// TIA Portal V16 export
// export: Created 2023-08-28T09:37:42.2517903Z, ExportSetting WithDefaults, DisplayName Totally Integrated Automation Portal, DisplayVersion V16 Update 6, DisplayName TIA Portal Version Control Interface, DisplayVersion V16 Update 2, DisplayName TIA Portal Openness, DisplayVersion V16 Update 6, DisplayName STEP 7 Professional, DisplayVersion V16 Update 6, DisplayName STEP 7 Safety, DisplayVersion V16, DisplayName WinCC Advanced, DisplayVersion V16 Update 6
FUNCTION_BLOCK "06_M_Main and auxiliary pump"   // FB9, LAD
TITLE = Funkcja ustalająca napęd wiodący i dodatkowe
{ S7_Optimized_Access := 'TRUE' }
AUTHOR : rtecmer
VERSION : 0.1
// Ustalanie silnika wiodącego i dodatkowego następuje po sprawdzeniu czy dany napęd załączony jes na falownik czy na sieć. Procedura rozpoczyna się od ustalenia napędu wiodącego.
// stored: AutoNumber true, IsIECCheckEnabled false, IsRetainMemResEnabled false, MemoryReserve 500, SetENOAutomatically false, UDAEnableTagReadback false
   VAR_IN_OUT
      set_Motor2 : Bool;   // pomocniczy bit ustawiania pompę dodatkową nr1
      set_Motor3 : Bool;   // pomocniczy bit ustawiania pompę dodatkową nr2
      set_Motor4 : Bool;   // pomocniczy bit ustawiania pompę dodatkową nr3
   END_VAR
   VAR_TEMP
      tmp_Res_Motor2 : Bool;   // pomocniczy bit kasowania znacznika dodatkowej nr1
      tmp_Res_Motor3 : Bool;   // pomocniczy bit kasowania znacznika dodatkowej nr2
      tmp_Res_Motor4 : Bool;   // pomocniczy bit kasowania znacznika dodatkowej nr3
   END_VAR
   VAR_TEMP   // added for the SCL form of the ladder/FBD networks
      _w1 : Bool;
      _w2 : Bool;
      _w3 : Bool;
      _w4 : Bool;
      _w5 : Bool;
      _w6 : Bool;
   END_VAR
BEGIN

REGION Network 1: Znacznik pompy wiodącej
   // M218.0 - bit ustalający pompy wiodącą . Przekazywany do zmiennych "IN" funkcji  "Control of   Inverters"
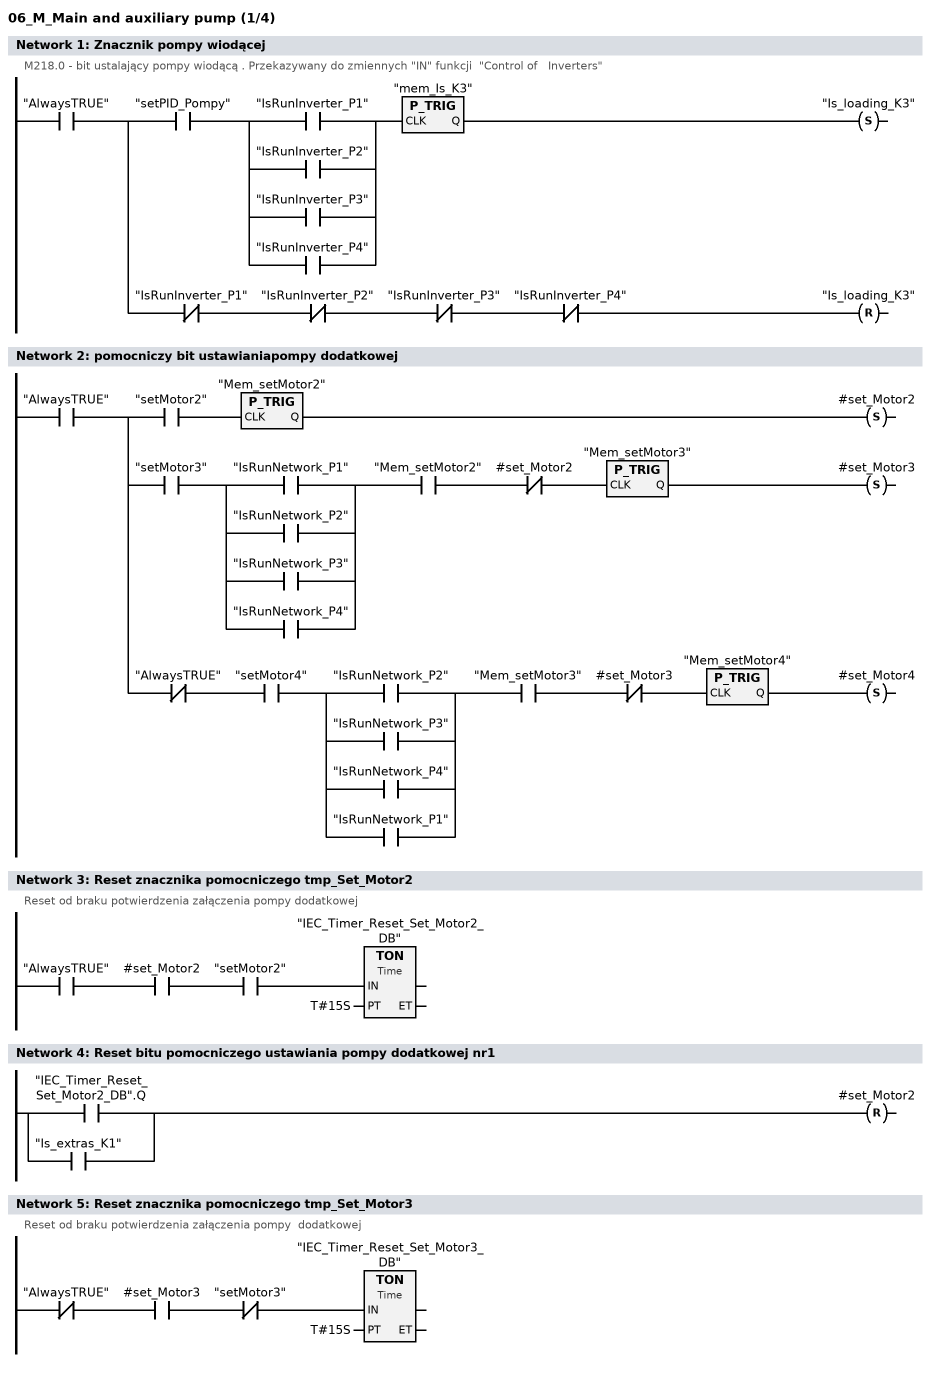
   RUNG wire#powerrail
      Contact( "AlwaysTRUE" )
      wire#w1
      Contact( "setPID_Pompy" )
      wire#w2
      Contact( "IsRunInverter_P1" )
      wire#w3
      P_Trig( "mem_Is_K3" )
      S_Coil( "Is_loading_K3" )
   END_RUNG
   RUNG wire#w2
      Contact( "IsRunInverter_P2" )
   END_RUNG wire#w3
   RUNG wire#w2
      Contact( "IsRunInverter_P3" )
   END_RUNG wire#w3
   RUNG wire#w2
      Contact( "IsRunInverter_P4" )
   END_RUNG wire#w3
   RUNG wire#w1
      I_Contact( "IsRunInverter_P1" )
      I_Contact( "IsRunInverter_P2" )
      I_Contact( "IsRunInverter_P3" )
      I_Contact( "IsRunInverter_P4" )
      R_Coil( "Is_loading_K3" )
   END_RUNG
   // the same network as SCL:
   #_w1 := "AlwaysTRUE" AND "setPID_Pompy" AND ("IsRunInverter_P1" OR "IsRunInverter_P2" OR "IsRunInverter_P3" OR "IsRunInverter_P4");
   #_w2 := #_w1 AND NOT "mem_Is_K3";   // rising edge
   "mem_Is_K3" := #_w1;
   IF #_w2 THEN "Is_loading_K3" := TRUE; END_IF;
   IF "AlwaysTRUE" AND NOT "IsRunInverter_P1" AND NOT "IsRunInverter_P2" AND NOT "IsRunInverter_P3" AND NOT "IsRunInverter_P4" THEN
       "Is_loading_K3" := FALSE;
   END_IF;
END_REGION

REGION Network 2: pomocniczy bit ustawianiapompy dodatkowej
   RUNG wire#powerrail
      Contact( "AlwaysTRUE" )
      wire#w1
      Contact( "setMotor2" )
      P_Trig( "Mem_setMotor2" )
      S_Coil( #set_Motor2 )
   END_RUNG
   RUNG wire#w1
      Contact( "setMotor3" )
      wire#w2
      Contact( "IsRunNetwork_P1" )
      wire#w3
      Contact( "Mem_setMotor2" )
      I_Contact( #set_Motor2 )
      P_Trig( "Mem_setMotor3" )
      S_Coil( #set_Motor3 )
   END_RUNG
   RUNG wire#w2
      Contact( "IsRunNetwork_P2" )
   END_RUNG wire#w3
   RUNG wire#w2
      Contact( "IsRunNetwork_P3" )
   END_RUNG wire#w3
   RUNG wire#w2
      Contact( "IsRunNetwork_P4" )
   END_RUNG wire#w3
   RUNG wire#w1
      I_Contact( "AlwaysTRUE" )
      Contact( "setMotor4" )
      wire#w4
      Contact( "IsRunNetwork_P2" )
      wire#w5
      Contact( "Mem_setMotor3" )
      I_Contact( #set_Motor3 )
      P_Trig( "Mem_setMotor4" )
      S_Coil( #set_Motor4 )
   END_RUNG
   RUNG wire#w4
      Contact( "IsRunNetwork_P3" )
   END_RUNG wire#w5
   RUNG wire#w4
      Contact( "IsRunNetwork_P4" )
   END_RUNG wire#w5
   RUNG wire#w4
      Contact( "IsRunNetwork_P1" )
   END_RUNG wire#w5
   // the same network as SCL:
   #_w1 := "AlwaysTRUE" AND "setMotor2";
   #_w2 := #_w1 AND NOT "Mem_setMotor2";   // rising edge
   "Mem_setMotor2" := #_w1;
   IF #_w2 THEN #set_Motor2 := TRUE; END_IF;
   #_w3 := "AlwaysTRUE" AND "setMotor3" AND ("IsRunNetwork_P1" OR "IsRunNetwork_P2" OR "IsRunNetwork_P3" OR "IsRunNetwork_P4") AND "Mem_setMotor2" AND NOT #set_Motor2;
   #_w4 := #_w3 AND NOT "Mem_setMotor3";   // rising edge
   "Mem_setMotor3" := #_w3;
   IF #_w4 THEN #set_Motor3 := TRUE; END_IF;
   #_w5 := "AlwaysTRUE" AND NOT "AlwaysTRUE" AND "setMotor4" AND ("IsRunNetwork_P2" OR "IsRunNetwork_P3" OR "IsRunNetwork_P4" OR "IsRunNetwork_P1") AND "Mem_setMotor3" AND NOT #set_Motor3;
   #_w6 := #_w5 AND NOT "Mem_setMotor4";   // rising edge
   "Mem_setMotor4" := #_w5;
   IF #_w6 THEN #set_Motor4 := TRUE; END_IF;
END_REGION

REGION Network 3: Reset znacznika pomocniczego tmp_Set_Motor2
   // Reset od braku potwierdzenia załączenia pompy dodatkowej
   RUNG wire#powerrail
      Contact( "AlwaysTRUE" )
      Contact( #set_Motor2 )
      Contact( "setMotor2" )
      { S7_Templates := "time_type := Time" } "IEC_Timer_Reset_Set_Motor2_DB".TON(pt := T#15S, et =>)
   END_RUNG
   // the same network as SCL:
   "IEC_Timer_Reset_Set_Motor2_DB".TON(IN := "AlwaysTRUE" AND #set_Motor2 AND "setMotor2", PT := T#15S);
END_REGION

REGION Network 4: Reset bitu pomocniczego ustawiania pompy dodatkowej nr1
   RUNG wire#powerrail
      Contact( "IEC_Timer_Reset_Set_Motor2_DB".Q )
      wire#w1
      R_Coil( #set_Motor2 )
   END_RUNG
   RUNG wire#powerrail
      Contact( "Is_extras_K1" )
   END_RUNG wire#w1
   // the same network as SCL:
   IF "IEC_Timer_Reset_Set_Motor2_DB".Q OR "Is_extras_K1" THEN #set_Motor2 := FALSE; END_IF;
END_REGION

REGION Network 5: Reset znacznika pomocniczego tmp_Set_Motor3
   // Reset od braku potwierdzenia załączenia pompy  dodatkowej
   RUNG wire#powerrail
      I_Contact( "AlwaysTRUE" )
      Contact( #set_Motor3 )
      I_Contact( "setMotor3" )
      { S7_Templates := "time_type := Time" } "IEC_Timer_Reset_Set_Motor3_DB".TON(pt := T#15S, et =>)
   END_RUNG
   // the same network as SCL:
   "IEC_Timer_Reset_Set_Motor3_DB".TON(IN := NOT "AlwaysTRUE" AND #set_Motor3 AND NOT "setMotor3", PT := T#15S);
END_REGION

REGION Network 6: Reset pomocniczego bit ustawianiapompy dodatkowej nr2
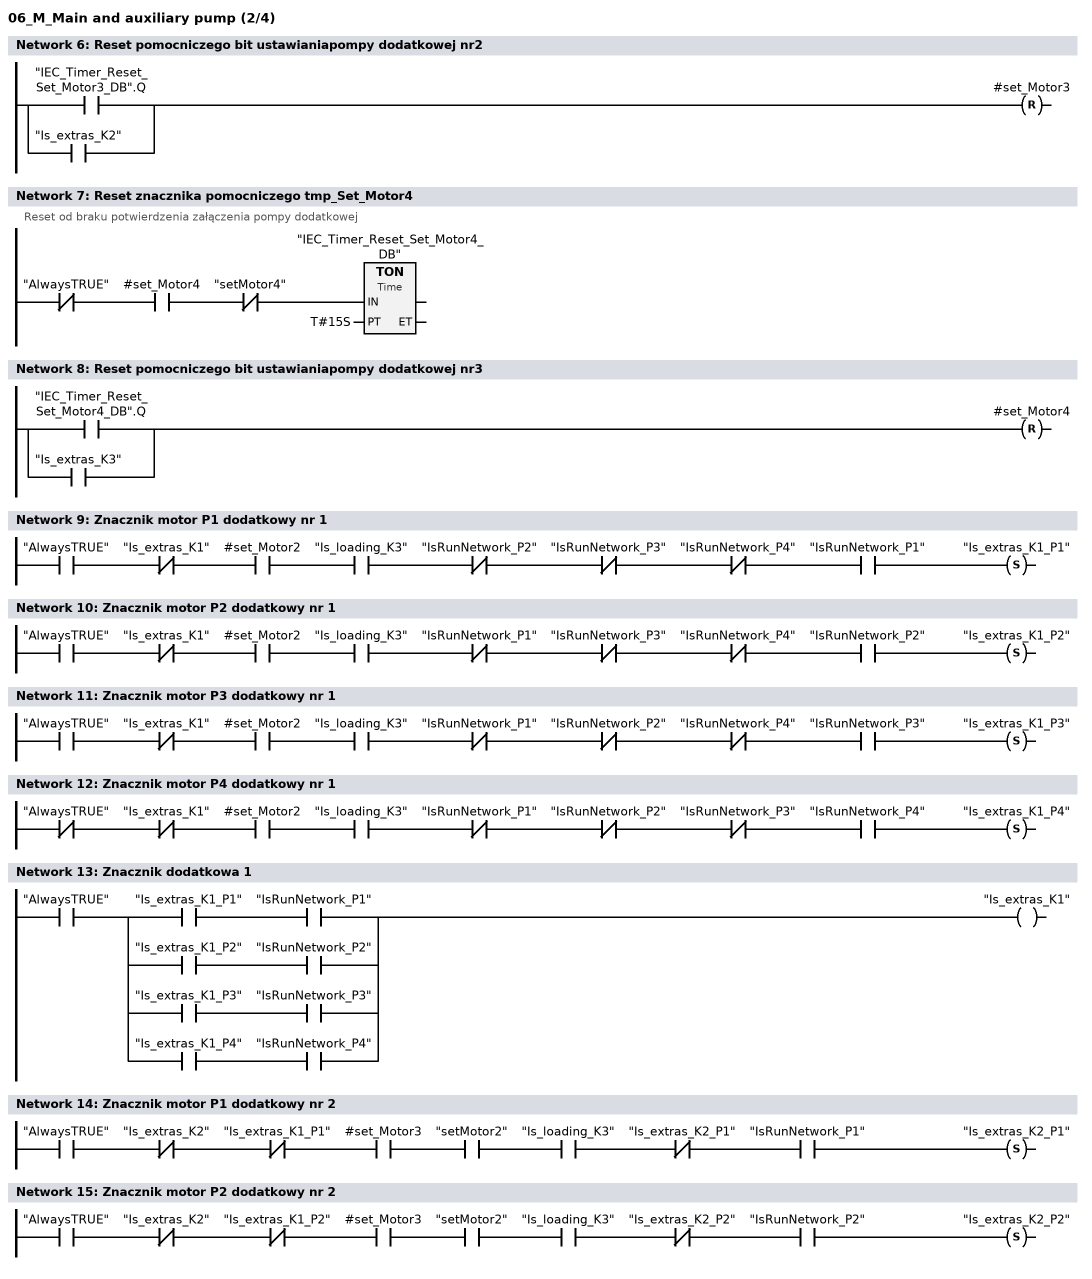
   RUNG wire#powerrail
      Contact( "IEC_Timer_Reset_Set_Motor3_DB".Q )
      wire#w1
      R_Coil( #set_Motor3 )
   END_RUNG
   RUNG wire#powerrail
      Contact( "Is_extras_K2" )
   END_RUNG wire#w1
   // the same network as SCL:
   IF "IEC_Timer_Reset_Set_Motor3_DB".Q OR "Is_extras_K2" THEN #set_Motor3 := FALSE; END_IF;
END_REGION

REGION Network 7: Reset znacznika pomocniczego tmp_Set_Motor4
   // Reset od braku potwierdzenia załączenia pompy dodatkowej
   RUNG wire#powerrail
      I_Contact( "AlwaysTRUE" )
      Contact( #set_Motor4 )
      I_Contact( "setMotor4" )
      { S7_Templates := "time_type := Time" } "IEC_Timer_Reset_Set_Motor4_DB".TON(pt := T#15S, et =>)
   END_RUNG
   // the same network as SCL:
   "IEC_Timer_Reset_Set_Motor4_DB".TON(IN := NOT "AlwaysTRUE" AND #set_Motor4 AND NOT "setMotor4", PT := T#15S);
END_REGION

REGION Network 8: Reset pomocniczego bit ustawianiapompy dodatkowej nr3
   RUNG wire#powerrail
      Contact( "IEC_Timer_Reset_Set_Motor4_DB".Q )
      wire#w1
      R_Coil( #set_Motor4 )
   END_RUNG
   RUNG wire#powerrail
      Contact( "Is_extras_K3" )
   END_RUNG wire#w1
   // the same network as SCL:
   IF "IEC_Timer_Reset_Set_Motor4_DB".Q OR "Is_extras_K3" THEN #set_Motor4 := FALSE; END_IF;
END_REGION

REGION Network 9: Znacznik motor P1 dodatkowy nr 1
   RUNG wire#powerrail
      Contact( "AlwaysTRUE" )
      I_Contact( "Is_extras_K1" )
      Contact( #set_Motor2 )
      Contact( "Is_loading_K3" )
      I_Contact( "IsRunNetwork_P2" )
      I_Contact( "IsRunNetwork_P3" )
      I_Contact( "IsRunNetwork_P4" )
      Contact( "IsRunNetwork_P1" )
      S_Coil( "Is_extras_K1_P1" )
   END_RUNG
   // the same network as SCL:
   IF "AlwaysTRUE" AND NOT "Is_extras_K1" AND #set_Motor2 AND "Is_loading_K3" AND NOT "IsRunNetwork_P2" AND NOT "IsRunNetwork_P3" AND NOT "IsRunNetwork_P4" AND "IsRunNetwork_P1" THEN
       "Is_extras_K1_P1" := TRUE;
   END_IF;
END_REGION

REGION Network 10: Znacznik motor P2 dodatkowy nr 1
   RUNG wire#powerrail
      Contact( "AlwaysTRUE" )
      I_Contact( "Is_extras_K1" )
      Contact( #set_Motor2 )
      Contact( "Is_loading_K3" )
      I_Contact( "IsRunNetwork_P1" )
      I_Contact( "IsRunNetwork_P3" )
      I_Contact( "IsRunNetwork_P4" )
      Contact( "IsRunNetwork_P2" )
      S_Coil( "Is_extras_K1_P2" )
   END_RUNG
   // the same network as SCL:
   IF "AlwaysTRUE" AND NOT "Is_extras_K1" AND #set_Motor2 AND "Is_loading_K3" AND NOT "IsRunNetwork_P1" AND NOT "IsRunNetwork_P3" AND NOT "IsRunNetwork_P4" AND "IsRunNetwork_P2" THEN
       "Is_extras_K1_P2" := TRUE;
   END_IF;
END_REGION

REGION Network 11: Znacznik motor P3 dodatkowy nr 1
   RUNG wire#powerrail
      Contact( "AlwaysTRUE" )
      I_Contact( "Is_extras_K1" )
      Contact( #set_Motor2 )
      Contact( "Is_loading_K3" )
      I_Contact( "IsRunNetwork_P1" )
      I_Contact( "IsRunNetwork_P2" )
      I_Contact( "IsRunNetwork_P4" )
      Contact( "IsRunNetwork_P3" )
      S_Coil( "Is_extras_K1_P3" )
   END_RUNG
   // the same network as SCL:
   IF "AlwaysTRUE" AND NOT "Is_extras_K1" AND #set_Motor2 AND "Is_loading_K3" AND NOT "IsRunNetwork_P1" AND NOT "IsRunNetwork_P2" AND NOT "IsRunNetwork_P4" AND "IsRunNetwork_P3" THEN
       "Is_extras_K1_P3" := TRUE;
   END_IF;
END_REGION

REGION Network 12: Znacznik motor P4 dodatkowy nr 1
   RUNG wire#powerrail
      I_Contact( "AlwaysTRUE" )
      I_Contact( "Is_extras_K1" )
      Contact( #set_Motor2 )
      Contact( "Is_loading_K3" )
      I_Contact( "IsRunNetwork_P1" )
      I_Contact( "IsRunNetwork_P2" )
      I_Contact( "IsRunNetwork_P3" )
      Contact( "IsRunNetwork_P4" )
      S_Coil( "Is_extras_K1_P4" )
   END_RUNG
   // the same network as SCL:
   IF NOT "AlwaysTRUE" AND NOT "Is_extras_K1" AND #set_Motor2 AND "Is_loading_K3" AND NOT "IsRunNetwork_P1" AND NOT "IsRunNetwork_P2" AND NOT "IsRunNetwork_P3" AND "IsRunNetwork_P4" THEN
       "Is_extras_K1_P4" := TRUE;
   END_IF;
END_REGION

REGION Network 13: Znacznik dodatkowa 1
   RUNG wire#powerrail
      Contact( "AlwaysTRUE" )
      wire#w1
      Contact( "Is_extras_K1_P1" )
      Contact( "IsRunNetwork_P1" )
      wire#w2
      Coil( "Is_extras_K1" )
   END_RUNG
   RUNG wire#w1
      Contact( "Is_extras_K1_P2" )
      Contact( "IsRunNetwork_P2" )
   END_RUNG wire#w2
   RUNG wire#w1
      Contact( "Is_extras_K1_P3" )
      Contact( "IsRunNetwork_P3" )
   END_RUNG wire#w2
   RUNG wire#w1
      Contact( "Is_extras_K1_P4" )
      Contact( "IsRunNetwork_P4" )
   END_RUNG wire#w2
   // the same network as SCL:
   "Is_extras_K1" := "AlwaysTRUE" AND (("Is_extras_K1_P1" AND "IsRunNetwork_P1") OR ("Is_extras_K1_P2" AND "IsRunNetwork_P2") OR ("Is_extras_K1_P3" AND "IsRunNetwork_P3") OR ("Is_extras_K1_P4" AND "IsRunNetwork_P4"));
END_REGION

REGION Network 14: Znacznik motor P1 dodatkowy nr 2
   RUNG wire#powerrail
      Contact( "AlwaysTRUE" )
      I_Contact( "Is_extras_K2" )
      I_Contact( "Is_extras_K1_P1" )
      Contact( #set_Motor3 )
      Contact( "setMotor2" )
      Contact( "Is_loading_K3" )
      I_Contact( "Is_extras_K2_P1" )
      Contact( "IsRunNetwork_P1" )
      S_Coil( "Is_extras_K2_P1" )
   END_RUNG
   // the same network as SCL:
   IF "AlwaysTRUE" AND NOT "Is_extras_K2" AND NOT "Is_extras_K1_P1" AND #set_Motor3 AND "setMotor2" AND "Is_loading_K3" AND NOT "Is_extras_K2_P1" AND "IsRunNetwork_P1" THEN
       "Is_extras_K2_P1" := TRUE;
   END_IF;
END_REGION

REGION Network 15: Znacznik motor P2 dodatkowy nr 2
   RUNG wire#powerrail
      Contact( "AlwaysTRUE" )
      I_Contact( "Is_extras_K2" )
      I_Contact( "Is_extras_K1_P2" )
      Contact( #set_Motor3 )
      Contact( "setMotor2" )
      Contact( "Is_loading_K3" )
      I_Contact( "Is_extras_K2_P2" )
      Contact( "IsRunNetwork_P2" )
      S_Coil( "Is_extras_K2_P2" )
   END_RUNG
   // the same network as SCL:
   IF "AlwaysTRUE" AND NOT "Is_extras_K2" AND NOT "Is_extras_K1_P2" AND #set_Motor3 AND "setMotor2" AND "Is_loading_K3" AND NOT "Is_extras_K2_P2" AND "IsRunNetwork_P2" THEN
       "Is_extras_K2_P2" := TRUE;
   END_IF;
END_REGION

REGION Network 16: Znacznik motor P3 dodatkowy nr 2
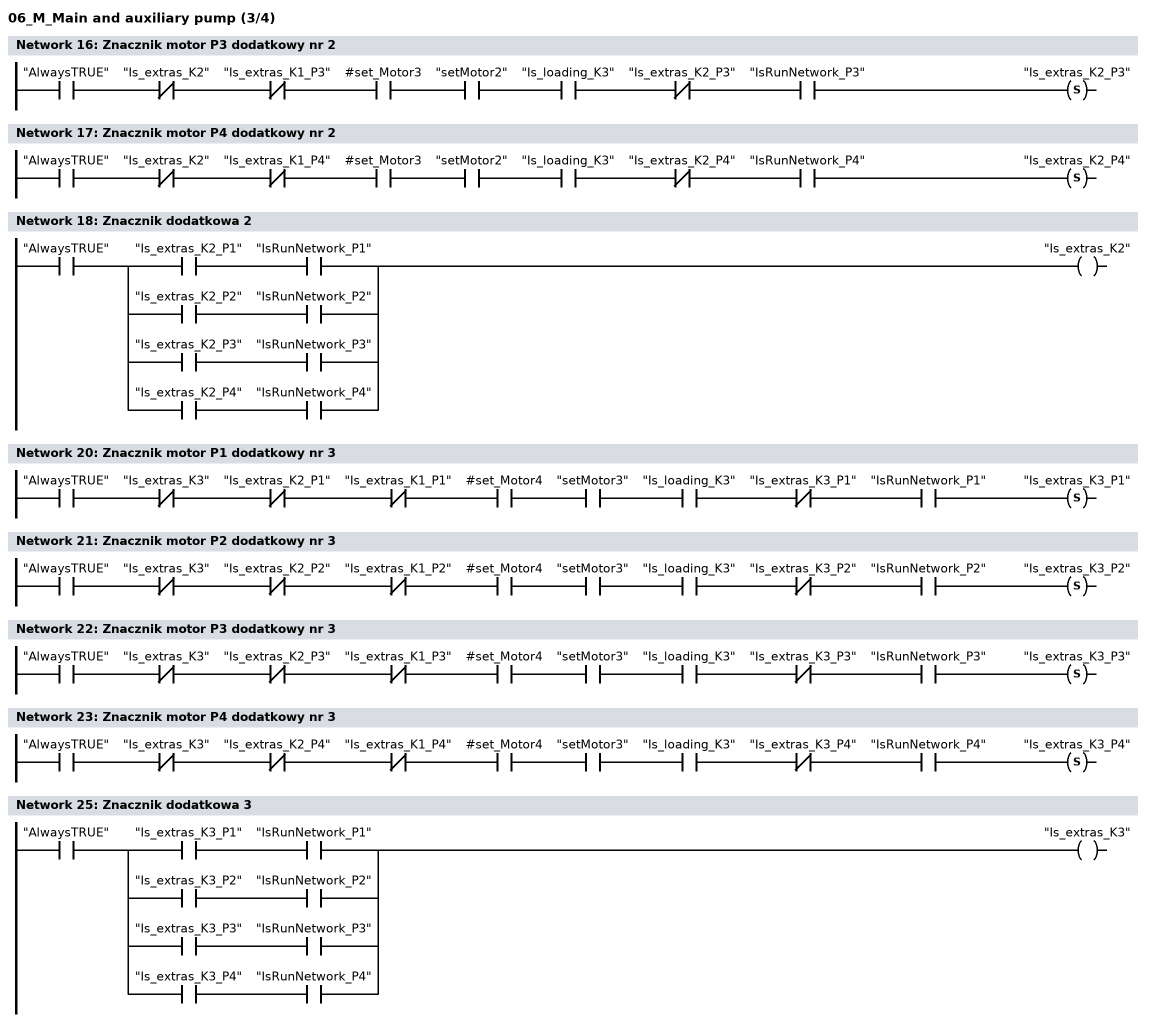
   RUNG wire#powerrail
      Contact( "AlwaysTRUE" )
      I_Contact( "Is_extras_K2" )
      I_Contact( "Is_extras_K1_P3" )
      Contact( #set_Motor3 )
      Contact( "setMotor2" )
      Contact( "Is_loading_K3" )
      I_Contact( "Is_extras_K2_P3" )
      Contact( "IsRunNetwork_P3" )
      S_Coil( "Is_extras_K2_P3" )
   END_RUNG
   // the same network as SCL:
   IF "AlwaysTRUE" AND NOT "Is_extras_K2" AND NOT "Is_extras_K1_P3" AND #set_Motor3 AND "setMotor2" AND "Is_loading_K3" AND NOT "Is_extras_K2_P3" AND "IsRunNetwork_P3" THEN
       "Is_extras_K2_P3" := TRUE;
   END_IF;
END_REGION

REGION Network 17: Znacznik motor P4 dodatkowy nr 2
   RUNG wire#powerrail
      Contact( "AlwaysTRUE" )
      I_Contact( "Is_extras_K2" )
      I_Contact( "Is_extras_K1_P4" )
      Contact( #set_Motor3 )
      Contact( "setMotor2" )
      Contact( "Is_loading_K3" )
      I_Contact( "Is_extras_K2_P4" )
      Contact( "IsRunNetwork_P4" )
      S_Coil( "Is_extras_K2_P4" )
   END_RUNG
   // the same network as SCL:
   IF "AlwaysTRUE" AND NOT "Is_extras_K2" AND NOT "Is_extras_K1_P4" AND #set_Motor3 AND "setMotor2" AND "Is_loading_K3" AND NOT "Is_extras_K2_P4" AND "IsRunNetwork_P4" THEN
       "Is_extras_K2_P4" := TRUE;
   END_IF;
END_REGION

REGION Network 18: Znacznik dodatkowa 2
   RUNG wire#powerrail
      Contact( "AlwaysTRUE" )
      wire#w1
      Contact( "Is_extras_K2_P1" )
      Contact( "IsRunNetwork_P1" )
      wire#w2
      Coil( "Is_extras_K2" )
   END_RUNG
   RUNG wire#w1
      Contact( "Is_extras_K2_P2" )
      Contact( "IsRunNetwork_P2" )
   END_RUNG wire#w2
   RUNG wire#w1
      Contact( "Is_extras_K2_P3" )
      Contact( "IsRunNetwork_P3" )
   END_RUNG wire#w2
   RUNG wire#w1
      Contact( "Is_extras_K2_P4" )
      Contact( "IsRunNetwork_P4" )
   END_RUNG wire#w2
   // the same network as SCL:
   "Is_extras_K2" := "AlwaysTRUE" AND (("Is_extras_K2_P1" AND "IsRunNetwork_P1") OR ("Is_extras_K2_P2" AND "IsRunNetwork_P2") OR ("Is_extras_K2_P3" AND "IsRunNetwork_P3") OR ("Is_extras_K2_P4" AND "IsRunNetwork_P4"));
END_REGION

REGION Network 20: Znacznik motor P1 dodatkowy nr 3
   RUNG wire#powerrail
      Contact( "AlwaysTRUE" )
      I_Contact( "Is_extras_K3" )
      I_Contact( "Is_extras_K2_P1" )
      I_Contact( "Is_extras_K1_P1" )
      Contact( #set_Motor4 )
      Contact( "setMotor3" )
      Contact( "Is_loading_K3" )
      I_Contact( "Is_extras_K3_P1" )
      Contact( "IsRunNetwork_P1" )
      S_Coil( "Is_extras_K3_P1" )
   END_RUNG
   // the same network as SCL:
   IF "AlwaysTRUE" AND NOT "Is_extras_K3" AND NOT "Is_extras_K2_P1" AND NOT "Is_extras_K1_P1" AND #set_Motor4 AND "setMotor3" AND "Is_loading_K3" AND NOT "Is_extras_K3_P1" AND "IsRunNetwork_P1" THEN
       "Is_extras_K3_P1" := TRUE;
   END_IF;
END_REGION

REGION Network 21: Znacznik motor P2 dodatkowy nr 3
   RUNG wire#powerrail
      Contact( "AlwaysTRUE" )
      I_Contact( "Is_extras_K3" )
      I_Contact( "Is_extras_K2_P2" )
      I_Contact( "Is_extras_K1_P2" )
      Contact( #set_Motor4 )
      Contact( "setMotor3" )
      Contact( "Is_loading_K3" )
      I_Contact( "Is_extras_K3_P2" )
      Contact( "IsRunNetwork_P2" )
      S_Coil( "Is_extras_K3_P2" )
   END_RUNG
   // the same network as SCL:
   IF "AlwaysTRUE" AND NOT "Is_extras_K3" AND NOT "Is_extras_K2_P2" AND NOT "Is_extras_K1_P2" AND #set_Motor4 AND "setMotor3" AND "Is_loading_K3" AND NOT "Is_extras_K3_P2" AND "IsRunNetwork_P2" THEN
       "Is_extras_K3_P2" := TRUE;
   END_IF;
END_REGION

REGION Network 22: Znacznik motor P3 dodatkowy nr 3
   RUNG wire#powerrail
      Contact( "AlwaysTRUE" )
      I_Contact( "Is_extras_K3" )
      I_Contact( "Is_extras_K2_P3" )
      I_Contact( "Is_extras_K1_P3" )
      Contact( #set_Motor4 )
      Contact( "setMotor3" )
      Contact( "Is_loading_K3" )
      I_Contact( "Is_extras_K3_P3" )
      Contact( "IsRunNetwork_P3" )
      S_Coil( "Is_extras_K3_P3" )
   END_RUNG
   // the same network as SCL:
   IF "AlwaysTRUE" AND NOT "Is_extras_K3" AND NOT "Is_extras_K2_P3" AND NOT "Is_extras_K1_P3" AND #set_Motor4 AND "setMotor3" AND "Is_loading_K3" AND NOT "Is_extras_K3_P3" AND "IsRunNetwork_P3" THEN
       "Is_extras_K3_P3" := TRUE;
   END_IF;
END_REGION

REGION Network 23: Znacznik motor P4 dodatkowy nr 3
   RUNG wire#powerrail
      Contact( "AlwaysTRUE" )
      I_Contact( "Is_extras_K3" )
      I_Contact( "Is_extras_K2_P4" )
      I_Contact( "Is_extras_K1_P4" )
      Contact( #set_Motor4 )
      Contact( "setMotor3" )
      Contact( "Is_loading_K3" )
      I_Contact( "Is_extras_K3_P4" )
      Contact( "IsRunNetwork_P4" )
      S_Coil( "Is_extras_K3_P4" )
   END_RUNG
   // the same network as SCL:
   IF "AlwaysTRUE" AND NOT "Is_extras_K3" AND NOT "Is_extras_K2_P4" AND NOT "Is_extras_K1_P4" AND #set_Motor4 AND "setMotor3" AND "Is_loading_K3" AND NOT "Is_extras_K3_P4" AND "IsRunNetwork_P4" THEN
       "Is_extras_K3_P4" := TRUE;
   END_IF;
END_REGION

REGION Network 25: Znacznik dodatkowa 3
   RUNG wire#powerrail
      Contact( "AlwaysTRUE" )
      wire#w1
      Contact( "Is_extras_K3_P1" )
      Contact( "IsRunNetwork_P1" )
      wire#w2
      Coil( "Is_extras_K3" )
   END_RUNG
   RUNG wire#w1
      Contact( "Is_extras_K3_P2" )
      Contact( "IsRunNetwork_P2" )
   END_RUNG wire#w2
   RUNG wire#w1
      Contact( "Is_extras_K3_P3" )
      Contact( "IsRunNetwork_P3" )
   END_RUNG wire#w2
   RUNG wire#w1
      Contact( "Is_extras_K3_P4" )
      Contact( "IsRunNetwork_P4" )
   END_RUNG wire#w2
   // the same network as SCL:
   "Is_extras_K3" := "AlwaysTRUE" AND (("Is_extras_K3_P1" AND "IsRunNetwork_P1") OR ("Is_extras_K3_P2" AND "IsRunNetwork_P2") OR ("Is_extras_K3_P3" AND "IsRunNetwork_P3") OR ("Is_extras_K3_P4" AND "IsRunNetwork_P4"));
END_REGION

REGION Network 26: pomocniczy bit ustawiania pompy dodatkowej nr1
   // Reset znacznika po udanym załączeniu pompy dodatkowej
   // Reset w wypadku braku pompy
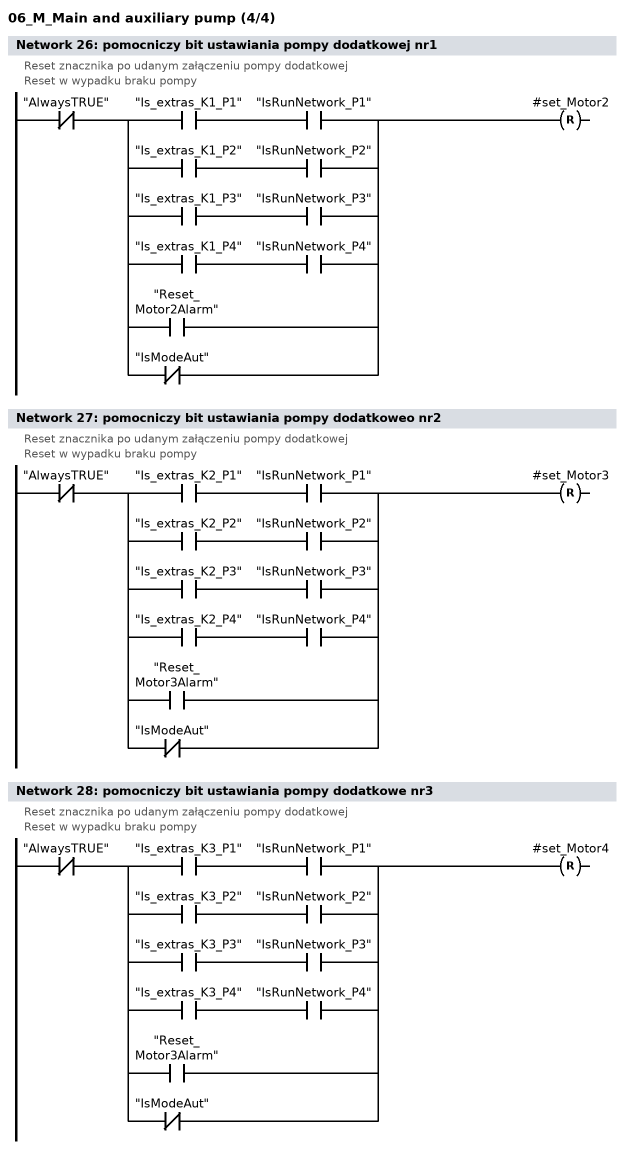
   RUNG wire#powerrail
      I_Contact( "AlwaysTRUE" )
      wire#w1
      Contact( "Is_extras_K1_P1" )
      Contact( "IsRunNetwork_P1" )
      wire#w2
      R_Coil( #set_Motor2 )
   END_RUNG
   RUNG wire#w1
      Contact( "Is_extras_K1_P2" )
      Contact( "IsRunNetwork_P2" )
   END_RUNG wire#w2
   RUNG wire#w1
      Contact( "Is_extras_K1_P3" )
      Contact( "IsRunNetwork_P3" )
   END_RUNG wire#w2
   RUNG wire#w1
      Contact( "Is_extras_K1_P4" )
      Contact( "IsRunNetwork_P4" )
   END_RUNG wire#w2
   RUNG wire#w1
      Contact( "Reset_Motor2Alarm" )
   END_RUNG wire#w2
   RUNG wire#w1
      I_Contact( "IsModeAut" )
   END_RUNG wire#w2
   // the same network as SCL:
   IF NOT "AlwaysTRUE" AND (("Is_extras_K1_P1" AND "IsRunNetwork_P1") OR ("Is_extras_K1_P2" AND "IsRunNetwork_P2") OR ("Is_extras_K1_P3" AND "IsRunNetwork_P3") OR ("Is_extras_K1_P4" AND "IsRunNetwork_P4") OR "Reset_Motor2Alarm" OR NOT "IsModeAut") THEN
       #set_Motor2 := FALSE;
   END_IF;
END_REGION

REGION Network 27: pomocniczy bit ustawiania pompy dodatkoweo nr2
   // Reset znacznika po udanym załączeniu pompy dodatkowej
   // Reset w wypadku braku pompy
   RUNG wire#powerrail
      I_Contact( "AlwaysTRUE" )
      wire#w1
      Contact( "Is_extras_K2_P1" )
      Contact( "IsRunNetwork_P1" )
      wire#w2
      R_Coil( #set_Motor3 )
   END_RUNG
   RUNG wire#w1
      Contact( "Is_extras_K2_P2" )
      Contact( "IsRunNetwork_P2" )
   END_RUNG wire#w2
   RUNG wire#w1
      Contact( "Is_extras_K2_P3" )
      Contact( "IsRunNetwork_P3" )
   END_RUNG wire#w2
   RUNG wire#w1
      Contact( "Is_extras_K2_P4" )
      Contact( "IsRunNetwork_P4" )
   END_RUNG wire#w2
   RUNG wire#w1
      Contact( "Reset_Motor3Alarm" )
   END_RUNG wire#w2
   RUNG wire#w1
      I_Contact( "IsModeAut" )
   END_RUNG wire#w2
   // the same network as SCL:
   IF NOT "AlwaysTRUE" AND (("Is_extras_K2_P1" AND "IsRunNetwork_P1") OR ("Is_extras_K2_P2" AND "IsRunNetwork_P2") OR ("Is_extras_K2_P3" AND "IsRunNetwork_P3") OR ("Is_extras_K2_P4" AND "IsRunNetwork_P4") OR "Reset_Motor3Alarm" OR NOT "IsModeAut") THEN
       #set_Motor3 := FALSE;
   END_IF;
END_REGION

REGION Network 28: pomocniczy bit ustawiania pompy dodatkowe nr3
   // Reset znacznika po udanym załączeniu pompy dodatkowej
   // Reset w wypadku braku pompy
   RUNG wire#powerrail
      I_Contact( "AlwaysTRUE" )
      wire#w1
      Contact( "Is_extras_K3_P1" )
      Contact( "IsRunNetwork_P1" )
      wire#w2
      R_Coil( #set_Motor4 )
   END_RUNG
   RUNG wire#w1
      Contact( "Is_extras_K3_P2" )
      Contact( "IsRunNetwork_P2" )
   END_RUNG wire#w2
   RUNG wire#w1
      Contact( "Is_extras_K3_P3" )
      Contact( "IsRunNetwork_P3" )
   END_RUNG wire#w2
   RUNG wire#w1
      Contact( "Is_extras_K3_P4" )
      Contact( "IsRunNetwork_P4" )
   END_RUNG wire#w2
   RUNG wire#w1
      Contact( "Reset_Motor3Alarm" )
   END_RUNG wire#w2
   RUNG wire#w1
      I_Contact( "IsModeAut" )
   END_RUNG wire#w2
   // the same network as SCL:
   IF NOT "AlwaysTRUE" AND (("Is_extras_K3_P1" AND "IsRunNetwork_P1") OR ("Is_extras_K3_P2" AND "IsRunNetwork_P2") OR ("Is_extras_K3_P3" AND "IsRunNetwork_P3") OR ("Is_extras_K3_P4" AND "IsRunNetwork_P4") OR "Reset_Motor3Alarm" OR NOT "IsModeAut") THEN
       #set_Motor4 := FALSE;
   END_IF;
END_REGION
END_FUNCTION_BLOCK
